FUNCTION_BLOCK CM_Sensor IMPLEMENTS  ITF_Sensor
VAR
	fb_mem : STRUCT_CM_Sensor;
END_VAR

(*
$$$$$$$$\                                                                   $$\       $$$$$$$$\                     $$\                                         $$\                     
$$  _____|                                                                  $$ |      $$  _____|                    \__|                                        \__|                    
$$ |   $$$$$$\   $$$$$$\  $$$$$$$\  $$\  $$\  $$\  $$$$$$\   $$$$$$\   $$$$$$$ |      $$ |      $$$$$$$\   $$$$$$\  $$\ $$$$$$$\   $$$$$$\   $$$$$$\   $$$$$$\  $$\ $$$$$$$\   $$$$$$\  
$$$$$\ \____$$\ $$  __$$\ $$  __$$\ $$ | $$ | $$ |$$  __$$\ $$  __$$\ $$  __$$ |      $$$$$\    $$  __$$\ $$  __$$\ $$ |$$  __$$\ $$  __$$\ $$  __$$\ $$  __$$\ $$ |$$  __$$\ $$  __$$\ 
$$  __|$$$$$$$ |$$ |  \__|$$ |  $$ |$$ | $$ | $$ |$$ /  $$ |$$ /  $$ |$$ /  $$ |      $$  __|   $$ |  $$ |$$ /  $$ |$$ |$$ |  $$ |$$$$$$$$ |$$$$$$$$ |$$ |  \__|$$ |$$ |  $$ |$$ /  $$ |
$$ |  $$  __$$ |$$ |      $$ |  $$ |$$ | $$ | $$ |$$ |  $$ |$$ |  $$ |$$ |  $$ |      $$ |      $$ |  $$ |$$ |  $$ |$$ |$$ |  $$ |$$   ____|$$   ____|$$ |      $$ |$$ |  $$ |$$ |  $$ |
$$ |  \$$$$$$$ |$$ |      $$ |  $$ |\$$$$$\$$$$  |\$$$$$$  |\$$$$$$  |\$$$$$$$ |      $$$$$$$$\ $$ |  $$ |\$$$$$$$ |$$ |$$ |  $$ |\$$$$$$$\ \$$$$$$$\ $$ |      $$ |$$ |  $$ |\$$$$$$$ |
\__|   \_______|\__|      \__|  \__| \_____\____/  \______/  \______/  \_______|      \________|\__|  \__| \____$$ |\__|\__|  \__| \_______| \_______|\__|      \__|\__|  \__| \____$$ |
                                                                                                          $$\   $$ |                                                          $$\   $$ |
                                                                                                          \$$$$$$  |                                                          \$$$$$$  |
                                                                                                           \______/                                                            \______/ 
*)

fb_mem.STS.Output := fb_mem.CS.Output;

//Zero all CS signals
fb_mem.CS.Auto		:= FALSE;
fb_mem.CS.Manueel 	:= FALSE;
fb_mem.CS.Output	:= FALSE;

//Zero all HMI signals
fb_mem.HMI.Auto		:= FALSE;
fb_mem.HMI.Manueel 	:= FALSE;
fb_mem.HMI.Output	:= FALSE;

PROPERTY Auto : BOOl
GET
AUTO := fb_mem.STS.Auto;
END_GET
SET
fb_mem.CS.Auto := AUTO;
END_SET
END_PROPERTY

METHOD FB_init : BOOL
VAR_INPUT
	bInitRetains : BOOL; // if TRUE, the retain variables are initialized (warm start / cold start)
	bInCopyCode : BOOL;  // if TRUE, the instance afterwards gets moved into the copy code (online change)
END_VAR
fb_mem.STS.Output := FALSE;
END_METHOD

PROPERTY Manueel : BOOl
GET
Manueel := fb_mem.STS.Manueel;
END_GET
SET
fb_mem.CS.Manueel :=  Manueel;
END_SET
END_PROPERTY

PROPERTY Output : BOOl
GET
Output := fb_mem.STS.Output;
END_GET
SET
fb_mem.CS.Output := Output;
END_SET
END_PROPERTY

PROPERTY Tag : STRING
GET
Tag := fb_mem.STS.Tag;
END_GET
END_PROPERTY

END_FUNCTION_BLOCK

(* stored: Version 1.1.0.1, ProductVersion 3.1.4024.12
   POU CM_Sensor: Id {9f7d1448-5df0-4be7-9ae0-ab06f7022e29}, SpecialFunc None
   Folder Methods: Id {d42d196e-9c2d-46ef-bb14-1c1bc71db29a}
   Folder Properties: Id {35572eb7-597e-443a-a59b-85d81a2710b8}
   Property Auto: Id {fe30e2d9-a541-4c1a-9d51-232d2f8d1608}
   Get Get: Id {26730b16-8f84-44b1-bfc9-49c9e6525e8e}
   Set Set: Id {7a2aa3d0-08ee-43bf-9080-aa8f53789611}
   Method FB_init: Id {5e5c01af-ec17-48b5-a03d-93d259206610}
   Property Manueel: Id {e8acbcdd-5600-4902-845c-c064adb43a10}
   Get Get: Id {65cbc6e7-537c-411a-aafb-2af3c7c38677}
   Set Set: Id {538b4d96-d5a8-4b52-88a1-43432404385c}
   Property Output: Id {7dcfaf3d-ebc2-4f7e-bc6f-c9179f9ed3fc}
   Get Get: Id {cc618e26-fe8e-4fe5-99d0-aa4f0666f865}
   Set Set: Id {582e1c4e-b2b9-45ae-8a2c-1b695346d955}
   Property Tag: Id {3a3e3dc0-b3ea-4d3c-93da-c8be1f8cfc53}
   Get Get: Id {8411c00c-d289-43d5-af20-e728117abe8d} *)
